(* Logix 5000 project; controller PLC_Safety vendor 1 type 14 code 148 rev 37.11; software revision 37.00 *)

TASK MainTask (continuous, watchdog 500 ms) : MainProgram
TASK SafetyTask (periodic, rate 20 ms, priority 10, watchdog 20 ms) : SafetyProgram

MODULES
   Local : vendor 1 type 14 code 148 (ICP 1, rev 37.11)
      Tarjeta_Ethernet : vendor 1 type 12 code 200 (ICP 0, Ethernet 10.12.143.10, rev 10.7, Input RPI 500 ms)
           Point_IO_Gabinete_6:2:I.1   // Push Button Gate 2 Reset
           Point_IO_Gabinete_6:2:I.2   // Push Button Gate 2 Open
         Kinetix_2 : vendor 1 type 37 code 48 (Ethernet 10.12.143.9, rev 7.1, MotionSync RPI 10 ms, MotionDiagnostics RPI 1 ms)
         Kinetix_1 : vendor 1 type 37 code 48 (Ethernet 10.12.143.8, rev 7.1, MotionDiagnostics RPI 1 ms, MotionSync RPI 10 ms)
         Cognex_3 : vendor 678 type 782 code 3585 (Ethernet 10.12.143.211, rev 1.1, StandardDataDriven RPI 20 ms)
         Fanuc_Brazo : vendor 8 type 140 code 34 (Ethernet 10.12.143.28, rev 2.4, StandardDataDriven RPI 20 ms)
              Fanuc_Brazo:I1.Input[2].4   // Input FANUC
              Fanuc_Brazo:I1.Input[3].0   // Input FANUC Rutina 5
              Fanuc_Brazo:I1.Input[3].1   // Input FANUC Rutina 6
              Fanuc_Brazo:I1.Input[3].2   // Input FANUC Rutina 7
              Fanuc_Brazo:O1.Output[0].3   // Cyle Stop - Abort
              Fanuc_Brazo:O1.Output[0]   // Fanuc Comands
              Fanuc_Brazo:O1.Output[2].0   // Strobe - Select
              Fanuc_Brazo:O1.Output[0].0   // Emergency Stop
              Fanuc_Brazo:O1.Output[0].1   // Hold
              Fanuc_Brazo:O1.Output[0].2   // Safe Speed
              Fanuc_Brazo:O1.Output[0].4   // Fault Reset
              Fanuc_Brazo:O1.Output[0].5   // Start
              Fanuc_Brazo:O1.Output[0].6   // Home
              Fanuc_Brazo:O1.Output[0].7   // Enable
              Fanuc_Brazo:O1.Output[1]   // Fanuc Routines
              Fanuc_Brazo:O1.Output[1].0   // No usar
              Fanuc_Brazo:O1.Output[1].1   // Routine 1 Base
              Fanuc_Brazo:O1.Output[1].2   // Routine 2 Centro
              Fanuc_Brazo:O1.Output[1].3   // Routine 3 Superior
              Fanuc_Brazo:O1.Output[1].4   // Routine 4 Assembly
              Fanuc_Brazo:O1.Output[2]   // Fanuc Strobe
         Fanuc_Delta : vendor 356 type 12 code 2 (Ethernet 10.12.143.47, rev 2.2, StandardDataDriven RPI 32 ms)
              Fanuc_Delta:I1.Input[0].1   // system ready
              Fanuc_Delta:I1.Input[0].0   // cmd enabled
              Fanuc_Delta:I1.Input[0].2   // prg running
              Fanuc_Delta:I1.Input[0].3   // prg paused
              Fanuc_Delta:I1.Input[0].4   // motion held
              Fanuc_Delta:I1.Input[0].5   // fault
              Fanuc_Delta:I1.Input[0].7   // tp enabled
              Fanuc_Delta:I1.Input[1].0   // batt alarm
              Fanuc_Delta:I1.Input[1].1   // busy
              Fanuc_Delta:I1.Input[1].2   // ack1
              Fanuc_Delta:I1.Input[1].3   // ack2
              Fanuc_Delta:I1.Input[1].4   // ack3
              Fanuc_Delta:I1.Input[1].5   // ack4
              Fanuc_Delta:I1.Input[1].6   // ack5
              Fanuc_Delta:I1.Input[1].7   // ack6
              Fanuc_Delta:I1.Input[2].0   // ack7
              Fanuc_Delta:I1.Input[2].1   // ack8
              Fanuc_Delta:I1.Input[2].2   // snack
              Fanuc_Delta:I1.Input[0].6   // at perch
              Fanuc_Delta:I1.Input[2].3   // reserved
              Fanuc_Delta:O1.Output[0].0   // IMSTP
              Fanuc_Delta:O1.Output[0].1   // hold
              Fanuc_Delta:O1.Output[0].2   // SFSPD
              Fanuc_Delta:O1.Output[0].3   // cycle stop
              Fanuc_Delta:O1.Output[0].4   // fault reset
              Fanuc_Delta:O1.Output[0].5   // start
              Fanuc_Delta:O1.Output[0].6   // Home
              Fanuc_Delta:O1.Output[0].7   // Enable
              Fanuc_Delta:O1.Output[1].0   // rsr1
              Fanuc_Delta:O1.Output[1].1   // rsr2
              Fanuc_Delta:O1.Output[1].2   // rsr3
              Fanuc_Delta:O1.Output[1].3   // rsr4
              Fanuc_Delta:O1.Output[1].4   // rsr5
              Fanuc_Delta:O1.Output[1].5   // rsr6
              Fanuc_Delta:O1.Output[1].6   // rsr7
              Fanuc_Delta:O1.Output[1].7   // rsr8
              Fanuc_Delta:O1.Output[2].0   // pns strobe
              Fanuc_Delta:O1.Output[2].1   // prod start
              Fanuc_Delta:O1.Output[2].5   // 22
              Fanuc_Delta:O1.Output[2].6   // 23
         Point_IO_Gabinete_3 : 1734-AENTR (Ethernet 10.12.143.42, rev 5.12, Output RPI 20 ms)
            Modulo_Input_Safety_3 : vendor 1 type 35 code 15 (PointIO 11, rev 2.2, Input RPI 10 ms)
                 Point_IO_Gabinete_3:11:I.Pt01Data   // Emergency Stop Conveyor 1 Normally Open
                 Point_IO_Gabinete_3:11:I.Pt00Data   // Emergency Stop Conveyor 1 Normally Close
                 Point_IO_Gabinete_3:11:I.Pt02Data   // SftyScanGab3 A (0=ObjDetec, 1=NoObjDetec)
                 Point_IO_Gabinete_3:11:I.Pt03Data   // SftyScanGab3 B (0=ObjDetec, 1=NoObjDetec)
            Modulo_Output_Safety_3 : vendor 1 type 35 code 16 (PointIO 12, rev 2.2, Input RPI 10 ms)
                 Point_IO_Gabinete_3:12:O.Pt01Data   // PowerFlex 1 Signal 2
                 Point_IO_Gabinete_3:12:O.Pt00Data   // PowerFlex 1 Signal 1
         Point_IO_Gabinete_1 : 1734-AENTR (Ethernet 10.12.143.40, rev 5.12, Output RPI 20 ms)
            Modulo_Output_Safety_1 : vendor 1 type 35 code 16 (PointIO 7, rev 2.2, Input RPI 10 ms)
                 Point_IO_Gabinete_1:7:O.Pt02Data   // GuardLock Gate 1
                 Point_IO_Gabinete_1:7:O.Pt01Data   // Kinetix 1 Signal 2
                 Point_IO_Gabinete_1:7:O.Pt00Data   // Kinetix 1 Signal 1
            Modulo_Input_Safety_1 : vendor 1 type 35 code 15 (PointIO 6, rev 2.2, Input RPI 10 ms)
                 Point_IO_Gabinete_1:6:I.Pt07Data   // Push Button Gate 1 Open
                 Point_IO_Gabinete_1:6:I.Pt05Data   // Guardlock Signal 2 Gate 1
                 Point_IO_Gabinete_1:6:I.Pt06Data   // Push Button Gate 1 Reset
                 Point_IO_Gabinete_1:6:I.Pt04Data   // GuardLock Signal 1 Gate 1
                 Point_IO_Gabinete_1:6:I.Pt01Data   // Emergency Stop 1 Normally Close
                 Point_IO_Gabinete_1:6:I.Pt00Data   // Emergency Stop 1 Normally Open
         Point_IO_Gabinete_2 : 1734-AENTR (Ethernet 10.12.143.41, rev 5.12, Output RPI 20 ms)   // Almacen Lado Derecho
            Modulo_Input_Safety_2 : vendor 1 type 35 code 15 (PointIO 6, rev 2.2, Input RPI 10 ms)
                 Point_IO_Gabinete_2:6:I.Pt06Data   // Push Button Process 2 Reset
                 Point_IO_Gabinete_2:6:I.Pt07Data   // Push Button Process 2 Start
                 Point_IO_Gabinete_2:6:I.Pt01Data   // Emergency Stop 2 Normally Close
                 Point_IO_Gabinete_2:6:I.Pt00Data   // Emergency Stop 2 Normally Open
            Modulo_Output_Safety_2 : vendor 1 type 35 code 16 (PointIO 7, rev 2.2, Input RPI 10 ms)
                 Point_IO_Gabinete_2:7:O.Pt01Data   // Kinetix 2 Signal 2
                 Point_IO_Gabinete_2:7:O.Pt00Data   // Kinetix 2 Signal 1
         Point_IO_Gabinete_4 : 1734-AENTR (Ethernet 10.12.143.43, rev 5.12, Output RPI 20 ms)   // Lado Izquierdo
            Modulo_Input_Safety_4 : vendor 1 type 35 code 15 (PointIO 11, rev 2.2, Input RPI 10 ms)
                 Point_IO_Gabinete_4:11:I.Pt02Data   // SftyScanGab4 A (0=ObjDetec, 1=NoObjDetec)
                 Point_IO_Gabinete_4:11:I.Pt03Data   // SftyScanGab4 B (0=ObjDetec, 1=NoObjDetec)
                 Point_IO_Gabinete_4:11:I.Pt01Data   // Emergency Stop Conveyor 2 Normally Open
                 Point_IO_Gabinete_4:11:I.Pt00Data   // Emergency Stop Conveyor 2 Normally Close
            Modulo_Output_Safety_4 : vendor 1 type 35 code 16 (PointIO 12, rev 2.2, Input RPI 10 ms)
                 Point_IO_Gabinete_4:12:O.Pt03Data   // Relay1 - ChB
                 Point_IO_Gabinete_4:12:O.Pt01Data   // Relay2 - ChB
                 Point_IO_Gabinete_4:12:O.Pt02Data   // Relay1 - ChA
                 Point_IO_Gabinete_4:12:O.Pt00Data   // Relay2 - ChA
                 Point_IO_Gabinete_4:12:O.Pt07Data   // PowerFlex 2 Signal 2
                 Point_IO_Gabinete_4:12:O.Pt06Data   // PowerFlex 2 Signal 1
         Point_IO_Gabinete_6 : 1734-AENTR (Ethernet 10.12.143.46, rev 5.11, Output RPI 20 ms)
            Modulo_Input_62 : 1734-IB8 (PointIO 2, rev 3.22)
            Modulo_Input_Safety_6 : vendor 1 type 35 code 15 (PointIO 4, rev 2.2, Input RPI 10 ms)
                 Point_IO_Gabinete_6:4:I.Pt01Data   // GuardLock Signal 2 Gate 2
                 Point_IO_Gabinete_6:4:I.Pt02Data   // Emergency Stop 3 Normally Close
                 Point_IO_Gabinete_6:4:I.Pt03Data   // Emergency Stop 3 Normally Open
                 Point_IO_Gabinete_6:4:I.Pt00Data   // GuardLock Signal 1 Gate 2
            Modulo_Output_Safety_6 : vendor 1 type 35 code 16 (PointIO 5, rev 2.2, Input RPI 10 ms)
                 Point_IO_Gabinete_6:5:O.Pt00Data   // GuardLock Gate 2
         PLC1 : vendor 1 type 14 code 235 (Ethernet 10.12.143.17, rev 37.11, $fc59bd35$ RPI 20 ms)
         PLC2 : vendor 1 type 14 code 235 (Ethernet 10.12.143.18, rev 37.11, $c2284200$ RPI 20 ms)
      @fcc730f7@:Partner : vendor 1 type 14 code 146 (ICP 2, rev 37.11)
END_MODULES

TYPE Auto_Data :
STRUCT
   Serial : STRING;
   Color : STRING;
   Peso : REAL;
   Llantas : DINT;
   Modo_Lujo : BOOL;
END_STRUCT
END_TYPE

VAR_GLOBAL   (* controller tags *)
   Axis_1 : AXIS_CIP_DRIVE;   // Storage 1
   Axis_2 : AXIS_CIP_DRIVE;   // Storage 2
   Data_From_PLC1 : DINT[20] := ([0] := 16781312);
   Data_From_PLC2 : DINT[20];
   Data_To_PLC1 : DINT[20] := ([0] := 1, [1] := 128); {produced}
        [0].13   // Tercera pieza recogida
        [0].12   // Segunda pieza recogida
        [0].11   // Primera pieza recogida
        [0].14   // Primera pieza para foto
        [0].15   // Segunda pieza para la foto
        [0].16   // Tercera pieza para la foto
   Data_To_PLC2 : DINT[20] := ([0] := 1, [2] := 1); {produced}
        [2].0   // E_stop_OK
   Display_Name : STRING;
   E_Stop_1_NC : ALIAS FOR Point_IO_Gabinete_1:6:I.Pt01Data;   // E Stop 1 Normally Close
   E_Stop_1_NO : ALIAS FOR Point_IO_Gabinete_1:6:I.Pt00Data;   // E Stop 1 Normally Open
   E_Stop_2_NC : ALIAS FOR Point_IO_Gabinete_2:6:I.Pt01Data;   // E Stop 2 Normally Close
   E_Stop_2_NO : ALIAS FOR Point_IO_Gabinete_2:6:I.Pt00Data;   // E Stop 2 Normally Open
   E_Stop_3_NC : ALIAS FOR Point_IO_Gabinete_6:4:I.Pt02Data;   // E Stop 3 Normally Close
   E_Stop_3_NO : ALIAS FOR Point_IO_Gabinete_6:4:I.Pt03Data;   // E Stop 3 Normally Open
   E_Stop_Conveyor_1_NC : ALIAS FOR Point_IO_Gabinete_3:11:I.Pt00Data;   // E Stop Conveyor 1 Normally Close
   E_Stop_Conveyor_1_NO : ALIAS FOR Point_IO_Gabinete_3:11:I.Pt01Data;   // E Stop Conveyor 1 Normally Open
   E_Stop_Conveyor_2_NC : ALIAS FOR Point_IO_Gabinete_4:11:I.Pt00Data;   // E Stop Conveyor 2 Normally Close
   E_Stop_Conveyor_2_NO : ALIAS FOR Point_IO_Gabinete_4:11:I.Pt01Data;   // E Stop Conveyor 2 Normally Open
   E_Stop_OK : BOOL := 1;
   Fanuc_E_Stop_SFTY : BOOL := 1;
   Fanuc_E_Stop_STD : BOOL := 1;
   Fanuc_Fault_Reset_SFTY : BOOL;
   Fanuc_Fault_Reset_STD : BOOL;
   Gate_1_Open_SFTY : ALIAS FOR Point_IO_Gabinete_1:6:I.Pt07Data;   // Push Button Gate 1 Open
   Gate_1_Reset_SFTY : ALIAS FOR Point_IO_Gabinete_1:6:I.Pt06Data;   // Push Button Gate 1 Reset
   Gate_2_Open_SFTY : BOOL;   // Push Button Gate 2 Open
   Gate_2_Open_STD : BOOL;   // Push Button Gate 2 Open
   Gate_2_Reset_SFTY : BOOL;   // Push Button Gate 2 Reset
   Gate_2_Reset_STD : BOOL;   // Push Button Gate 2 Reset
   Manual_SFTY : BOOL := 1;
   Manual_STD : BOOL := 1;
   Motion : MOTION_GROUP;
   Process_1_Reset_SFTY : BOOL;   // Push Button Process 1 Reset
   Process_1_Reset_STD : BOOL;   // Push Button Process 1 Reset
   Process_2_Reset_SFTY : ALIAS FOR Point_IO_Gabinete_2:6:I.Pt06Data;   // Push Button Process 2 Reset
   Process_2_Start_SFTY : ALIAS FOR Point_IO_Gabinete_2:6:I.Pt07Data;   // Push Button Porcess 2 Start
   Reset_General : BOOL;
   S1_Height_1 : BOOL;
   S1_Height_2 : BOOL;
   S1_Height_3 : BOOL;
   S1_Height_4 : BOOL;
   S1_Height_5 : BOOL;
   S1_Height_6 : BOOL;
   S1_Height_Conveyor_1 : BOOL;
   S1_Height_Conveyor_2 : BOOL;
   S1_Storage_On : BOOL;
   Safety_OK : BOOL := 1;
   Start_Button_1_Squence : BOOL;
END_VAR

PROGRAM MainProgram   (* main routine R00_Main_Routine *)
VAR
   Assembly_Step : DINT;
   Contador_num_pza : COUNTER;
   Contador_pza_aprove : COUNTER := (CU := 1, DN := 1);
   Contador_pza_rechazada : COUNTER := (DN := 1);
   Counter_Parts : COUNTER := (ACC := 2, CU := 1, DN := 1);   // Trazabilidad
   Done_cicle : BOOL;
   Error_Cam : DINT;
   FANUC_R1 : BOOL := 1;
   FANUC_R2 : BOOL;
   FANUC_R3 : BOOL;
   FANUC_R4 : BOOL;
   Fanuc_Strobe : BOOL;
   HMI_Cognex_1 : DINT;   // HMI
   HMI_Cognex_2 : DINT;   // HMI
   HMI_Cognex_medio : DINT;   // HMI
   HMI_Fanucbrazo : DINT := 516;   // HMI
   HMI_Fanucdelta : DINT := 516;   // HMI
   HMI_Fcognex1 : BOOL;   // HMI
   HMI_Fcognex2 : BOOL;   // HMI
   HMI_Fcognexmedio : BOOL;   // HMI
   HMI_Ffanucbrazo : BOOL := 1;   // HMI
   HMI_Ffanucdelta : BOOL := 1;   // HMI
   HMI_Fplc1 : BOOL;   // HMI
   HMI_Fplc2 : BOOL;   // HMI
   HMI_Fplcseguridad : BOOL;   // HMI
   HMI_kinetix1 : BOOL;   // HMI
   HMI_kinetix2 : BOOL;
   HMI_Kinetix_1 : DINT;   // HMI
   HMI_Kinetix_2 : DINT;
   HMI_PLC1 : DINT;   // HMI
   HMI_PLC2 : DINT;   // HMI
   HMI_PLC_Seguridad : DINT;   // HMI
   HMI_PointIO1 : BOOL;   // HMI
   HMI_PointIO2 : BOOL;
   HMI_PointIO3 : BOOL;
   HMI_PointIO4 : BOOL;
   HMI_PointIO6 : BOOL;
   HMI_PointIO_1 : DINT;   // HMI
   HMI_PointIO_2 : DINT;
   HMI_PointIO_3 : DINT;
   HMI_PointIO_4 : DINT;
   HMI_PointIO_6 : DINT;
   HMI_R_Axis_Y_Negative : BOOL;
   HMI_R_Axis_Y_Positive : BOOL;
   HMI_R_cognex1 : BOOL := 1;
   HMI_R_cognex2 : BOOL;
   HMI_R_con2OFF : BOOL;
   HMI_R_con2ON : BOOL;
   HMI_R_Conveyor_OFF : BOOL;
   HMI_R_Conveyor_ON : BOOL;
   HMI_R_Gripper_Close : BOOL;
   HMI_R_Gripper_Open : BOOL;
   HMI_R_Height_4_1 : BOOL;
   HMI_R_Height_4_2 : BOOL;
   HMI_R_Height_5_1 : BOOL;
   HMI_R_Height_5_2 : BOOL;
   HMI_R_Height_6_1 : BOOL;
   HMI_R_Height_6_2 : BOOL;
   HMI_R_lane1 : BOOL;
   HMI_R_lane1_c2 : BOOL;
   HMI_R_lane2 : BOOL;
   HMI_R_lane2_c2 : BOOL;
   HMI_R_onoff : BOOL := 1;
   HMI_R_PF1 : BOOL;
   HMI_R_PF2 : BOOL;
   HMI_R_pis0 : BOOL;
   HMI_R_pis1 : BOOL;
   HMI_R_pis2 : BOOL;
   HMI_R_pis3 : BOOL;
   HMI_R_pis4 : BOOL;
   HMI_R_pis5 : BOOL;
   HMI_R_pis6 : BOOL;
   HMI_R_pis7 : BOOL;
   HMI_R_pis8 : BOOL;
   HMI_R_pis9 : BOOL;
   HMI_R_Turn_Conveyor : BOOL;
   HMI_R_Turn_Storage : BOOL;
   HMI_S_Axis_Y_Negative : BOOL;
   HMI_S_Axis_Y_Positive : BOOL;
   HMI_S_cognex1 : BOOL := 1;
   HMI_S_cognex2 : BOOL;
   HMI_S_con2Off : BOOL;
   HMI_S_con2ON : BOOL;
   HMI_S_Conveyor_OFF : BOOL;
   HMI_S_Conveyor_ON : BOOL;
   HMI_S_Gripper_Close : BOOL;
   HMI_S_Gripper_Open : BOOL;
   HMI_S_Height_4_1 : BOOL;
   HMI_S_Height_4_2 : BOOL;
   HMI_S_Height_5_1 : BOOL;
   HMI_S_Height_5_2 : BOOL;
   HMI_S_Height_6_1 : BOOL;
   HMI_S_Height_6_2 : BOOL;
   HMI_S_lane1 : BOOL;
   HMI_S_lane1_c2 : BOOL;
   HMI_S_lane2 : BOOL;
   HMI_S_lane2_c2 : BOOL;
   HMI_S_onoff : BOOL := 1;
   HMI_S_PF1 : BOOL;
   HMI_S_PF2 : BOOL;
   HMI_S_pis0 : BOOL;
   HMI_S_pis1 : BOOL;
   HMI_S_pis2 : BOOL;
   HMI_S_pis3 : BOOL;
   HMI_S_pis4 : BOOL;
   HMI_S_pis5 : BOOL;
   HMI_S_pis6 : BOOL;
   HMI_S_pis7 : BOOL;
   HMI_S_pis8 : BOOL;
   HMI_S_pis9 : BOOL;
   HMI_S_Turn_Conveyor : BOOL;
   HMI_S_Turn_Storage : BOOL;
   HMI_Switch1 : BOOL;
   HMI_Switch2 : BOOL;
   HMI_Switch3 : BOOL := 1;
   HMI_Switch4 : BOOL;
   HMI_Switch5 : BOOL := 1;
   OSF_Fault_Reset_Fanuc : BOOL;
   Part : REAL := 1.0;
   Piece_Approved : BOOL := 1;
   Piece_Base : BOOL := 1;
   Piece_Coil : BOOL;
   Piece_Rejected : BOOL;
   Piece_Upper : BOOL;
   Process_Result : BOOL;
   Result_OneShot : BOOL;
   S1_Height_4_Number_2 : BOOL;
   S1_Height_5_Number_2 : BOOL;
   S1_Height_6_Number_2 : BOOL;
   S1_MAM_Height_1 : MOTION_INSTRUCTION := (FLAGS := 33554432);
   S1_MAM_Height_2 : MOTION_INSTRUCTION := (FLAGS := 33554432);
   S1_MAM_Height_3 : MOTION_INSTRUCTION := (FLAGS := 33554432);
   S1_MAM_Height_4 : MOTION_INSTRUCTION := (FLAGS := 33554432);
   S1_MAM_Height_4_Number_2 : MOTION_INSTRUCTION := (FLAGS := 33554432);
   S1_MAM_Height_5 : MOTION_INSTRUCTION := (FLAGS := 33554432);
   S1_MAM_Height_5_Number_2 : MOTION_INSTRUCTION := (FLAGS := 33554432);
   S1_MAM_Height_6 : MOTION_INSTRUCTION := (FLAGS := 33554432);
   S1_MAM_Height_6_Number_2 : MOTION_INSTRUCTION := (FLAGS := 33554432);
   S1_MAM_Height_Conveyor_1 : MOTION_INSTRUCTION := (FLAGS := 33554432);
   S1_MAM_Height_Conveyor_2 : MOTION_INSTRUCTION := (FLAGS := 33554432);
   S1_MSO_Storage : MOTION_INSTRUCTION := (FLAGS := 33554432);
   S1_Sensor_Height_1 : BOOL;
   S1_Sensor_Height_2 : BOOL;
   S1_Sensor_Height_3 : BOOL;
   S1_Sensor_Height_4 : BOOL;
   S1_Sensor_Height_4_Number_2 : BOOL;
   S1_Sensor_Height_5 : BOOL;
   S1_Sensor_Height_5_Number_2 : BOOL;
   S1_Sensor_Height_6 : BOOL;
   S1_Sensor_Height_6_Number_2 : BOOL;
   S1_Sensor_Height_Conveyor_1 : BOOL;
   S1_Sensor_Height_Conveyor_2 : BOOL;
   S2_Height_1 : BOOL;
   S2_Height_2 : BOOL;
   S2_Height_3 : BOOL;
   S2_Height_4 : BOOL;
   S2_Height_4_Number_2 : BOOL;
   S2_Height_5 : BOOL;
   S2_Height_5_Number_2 : BOOL;
   S2_Height_6 : BOOL;
   S2_Height_Conveyor_1 : BOOL;
   S2_Height_Conveyor_2 : BOOL;
   S2_MAM_Height_1 : MOTION_INSTRUCTION;
   S2_MAM_Height_2 : MOTION_INSTRUCTION;
   S2_MAM_Height_3 : MOTION_INSTRUCTION;
   S2_MAM_Height_4 : MOTION_INSTRUCTION;
   S2_MAM_Height_4_Number_2 : MOTION_INSTRUCTION;
   S2_MAM_Height_5 : MOTION_INSTRUCTION;
   S2_MAM_Height_5_Number_2 : MOTION_INSTRUCTION;
   S2_MAM_Height_6 : MOTION_INSTRUCTION;
   S2_MAM_Height_Conveyor_1 : MOTION_INSTRUCTION;
   S2_MAM_Height_Conveyor_2 : MOTION_INSTRUCTION;
   S2_MSO_Storage : MOTION_INSTRUCTION;
   S2_Sensor_Height_1 : BOOL;
   S2_Sensor_Height_2 : BOOL;
   S2_Sensor_Height_3 : BOOL;
   S2_Sensor_Height_4 : BOOL;
   S2_Sensor_Height_5 : BOOL;
   S2_Sensor_Height_6 : BOOL;
   S2_Sensor_Height_Conveyor_1 : BOOL;
   S2_Sensor_Height_Conveyor_2 : BOOL;
   S2_Storage_On : BOOL;
   Sensor_FANUC_R1 : BOOL;
   Sensor_FANUC_R2 : BOOL;
   Sensor_FANUC_R3 : BOOL;
   Sensor_FANUC_R4 : BOOL;
   Start_Button_1_Secuencia : BOOL;
   Start_Button_2_Secuencia : BOOL;
   Start_Button_3_Secuencia : BOOL;
   Stop_general : BOOL;
   Trigger_Cognex_3 : BOOL;
END_VAR

ROUTINE HMI_Manual_Safety   (* ladder *)
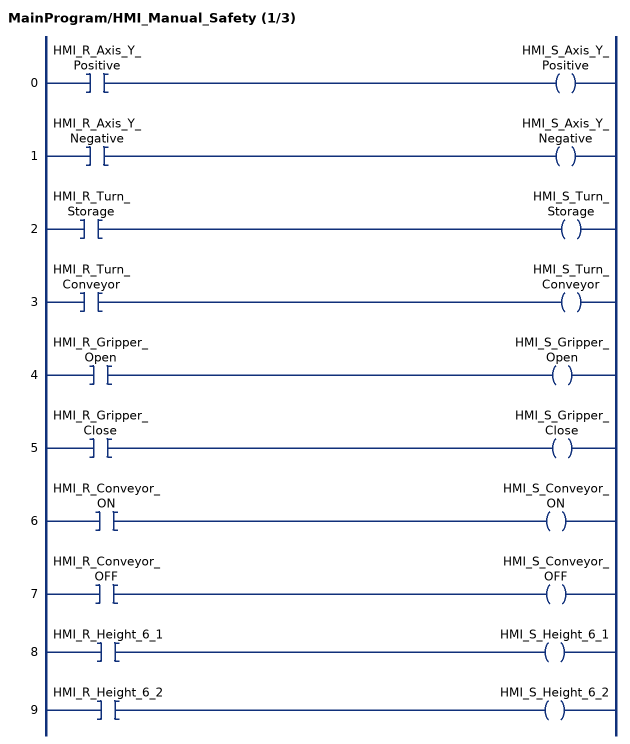
   0: XIC(HMI_R_Axis_Y_Positive)OTE(HMI_S_Axis_Y_Positive);
   1: XIC(HMI_R_Axis_Y_Negative)OTE(HMI_S_Axis_Y_Negative);
   2: XIC(HMI_R_Turn_Storage)OTE(HMI_S_Turn_Storage);
   3: XIC(HMI_R_Turn_Conveyor)OTE(HMI_S_Turn_Conveyor);
   4: XIC(HMI_R_Gripper_Open)OTE(HMI_S_Gripper_Open);
   5: XIC(HMI_R_Gripper_Close)OTE(HMI_S_Gripper_Close);
   6: XIC(HMI_R_Conveyor_ON)OTE(HMI_S_Conveyor_ON);
   7: XIC(HMI_R_Conveyor_OFF)OTE(HMI_S_Conveyor_OFF);
   8: XIC(HMI_R_Height_6_1)OTE(HMI_S_Height_6_1);
   9: XIC(HMI_R_Height_6_2)OTE(HMI_S_Height_6_2);
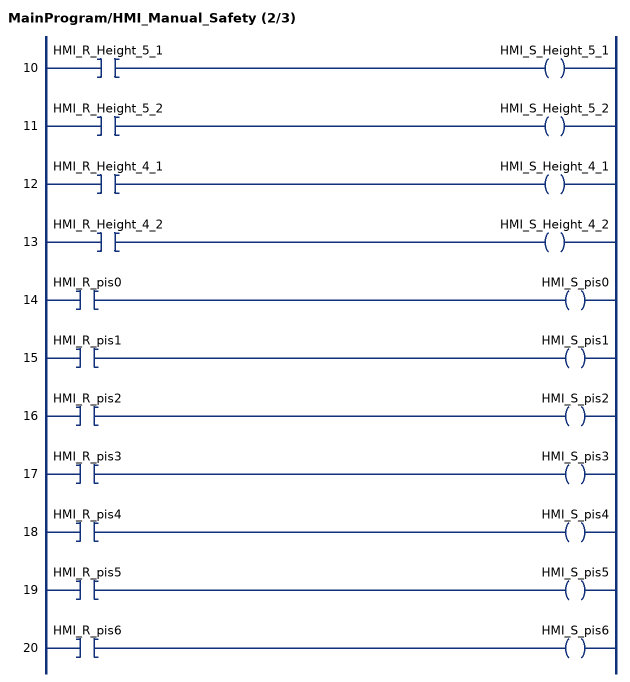
   10: XIC(HMI_R_Height_5_1)OTE(HMI_S_Height_5_1);
   11: XIC(HMI_R_Height_5_2)OTE(HMI_S_Height_5_2);
   12: XIC(HMI_R_Height_4_1)OTE(HMI_S_Height_4_1);
   13: XIC(HMI_R_Height_4_2)OTE(HMI_S_Height_4_2);
   14: XIC(HMI_R_pis0)OTE(HMI_S_pis0);
   15: XIC(HMI_R_pis1)OTE(HMI_S_pis1);
   16: XIC(HMI_R_pis2)OTE(HMI_S_pis2);
   17: XIC(HMI_R_pis3)OTE(HMI_S_pis3);
   18: XIC(HMI_R_pis4)OTE(HMI_S_pis4);
   19: XIC(HMI_R_pis5)OTE(HMI_S_pis5);
   20: XIC(HMI_R_pis6)OTE(HMI_S_pis6);
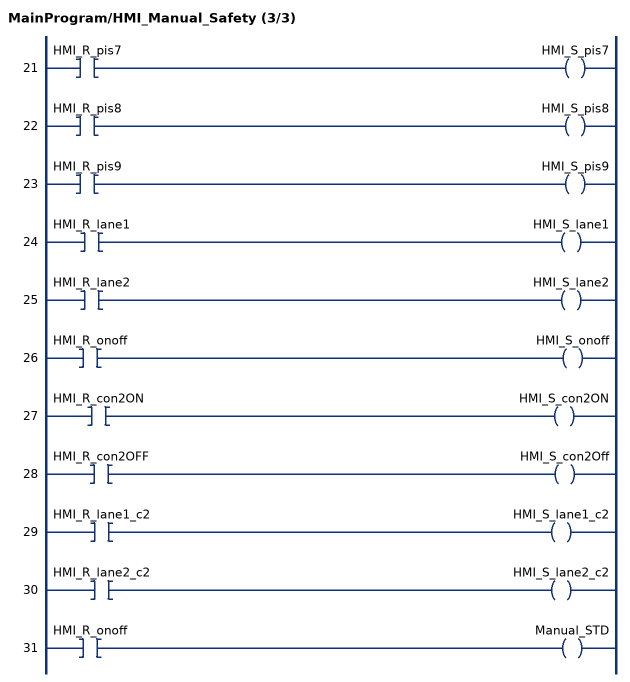
   21: XIC(HMI_R_pis7)OTE(HMI_S_pis7);
   22: XIC(HMI_R_pis8)OTE(HMI_S_pis8);
   23: XIC(HMI_R_pis9)OTE(HMI_S_pis9);
   24: XIC(HMI_R_lane1)OTE(HMI_S_lane1);
   25: XIC(HMI_R_lane2)OTE(HMI_S_lane2);
   26: XIC(HMI_R_onoff)OTE(HMI_S_onoff);
   27: XIC(HMI_R_con2ON)OTE(HMI_S_con2ON);
   28: XIC(HMI_R_con2OFF)OTE(HMI_S_con2Off);
   29: XIC(HMI_R_lane1_c2)OTE(HMI_S_lane1_c2);
   30: XIC(HMI_R_lane2_c2)OTE(HMI_S_lane2_c2);
   31: XIC(HMI_R_onoff)OTE(Manual_STD);
END_ROUTINE

ROUTINE R00_Main_Routine   (* ladder *)
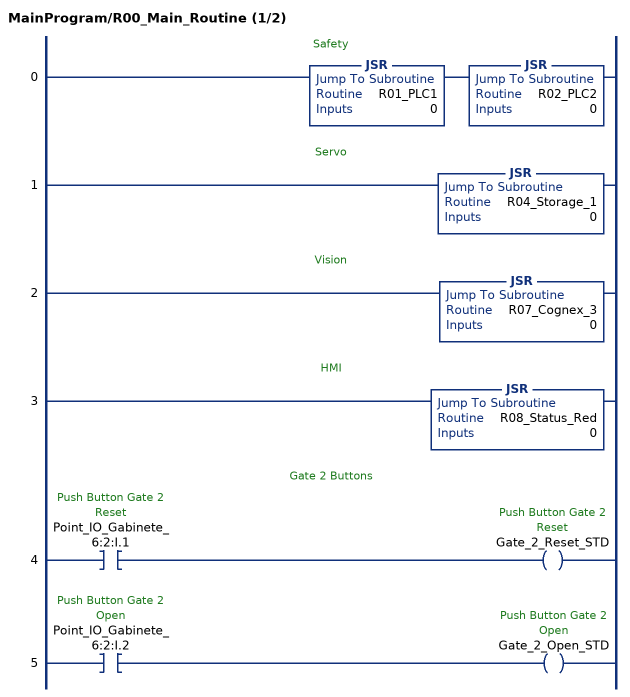
   // Safety
   0: JSR(R01_PLC1,0)JSR(R02_PLC2,0);
   // Servo
   1: JSR(R04_Storage_1,0);
   // Vision
   2: JSR(R07_Cognex_3,0);
   // HMI
   3: JSR(R08_Status_Red,0);
   // Gate 2 Buttons
   4: XIC(Point_IO_Gabinete_6:2:I.1)OTE(Gate_2_Reset_STD);
   5: XIC(Point_IO_Gabinete_6:2:I.2)OTE(Gate_2_Open_STD);
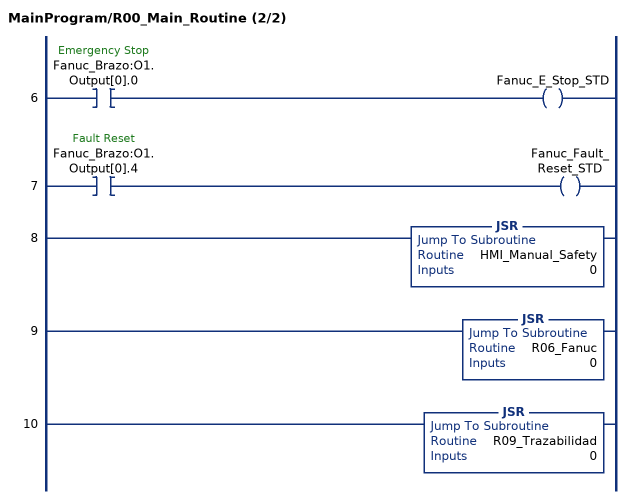
   6: XIC(Fanuc_Brazo:O1.Output[0].0)OTE(Fanuc_E_Stop_STD);
   7: XIC(Fanuc_Brazo:O1.Output[0].4)OTE(Fanuc_Fault_Reset_STD);
   8: JSR(HMI_Manual_Safety,0);
   9: JSR(R06_Fanuc,0);
   10: JSR(R09_Trazabilidad,0);
END_ROUTINE

ROUTINE R01_PLC1   (* ladder *)
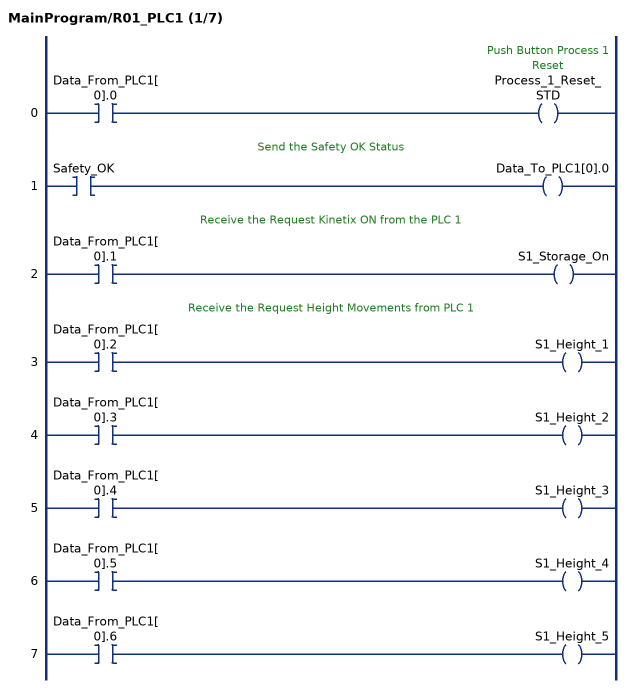
   0: XIC(Data_From_PLC1[0].0)OTE(Process_1_Reset_STD);
   // Send the Safety OK Status
   1: XIC(Safety_OK)OTE(Data_To_PLC1[0].0);
   // Receive the Request Kinetix ON from the PLC 1
   2: XIC(Data_From_PLC1[0].1)OTE(S1_Storage_On);
   // Receive the Request Height Movements from PLC 1
   3: XIC(Data_From_PLC1[0].2)OTE(S1_Height_1);
   4: XIC(Data_From_PLC1[0].3)OTE(S1_Height_2);
   5: XIC(Data_From_PLC1[0].4)OTE(S1_Height_3);
   6: XIC(Data_From_PLC1[0].5)OTE(S1_Height_4);
   7: XIC(Data_From_PLC1[0].6)OTE(S1_Height_5);
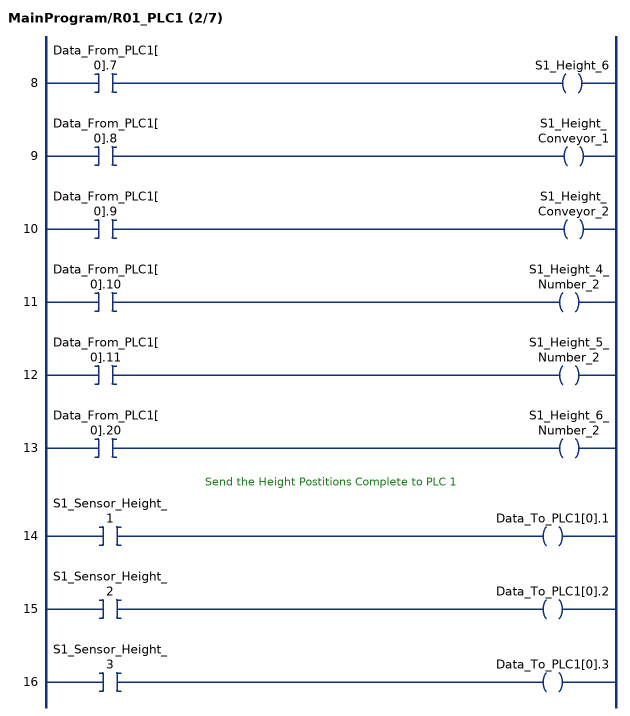
   8: XIC(Data_From_PLC1[0].7)OTE(S1_Height_6);
   9: XIC(Data_From_PLC1[0].8)OTE(S1_Height_Conveyor_1);
   10: XIC(Data_From_PLC1[0].9)OTE(S1_Height_Conveyor_2);
   11: XIC(Data_From_PLC1[0].10)OTE(S1_Height_4_Number_2);
   12: XIC(Data_From_PLC1[0].11)OTE(S1_Height_5_Number_2);
   13: XIC(Data_From_PLC1[0].20)OTE(S1_Height_6_Number_2);
   // Send the Height Postitions Complete to PLC 1
   14: XIC(S1_Sensor_Height_1)OTE(Data_To_PLC1[0].1);
   15: XIC(S1_Sensor_Height_2)OTE(Data_To_PLC1[0].2);
   16: XIC(S1_Sensor_Height_3)OTE(Data_To_PLC1[0].3);
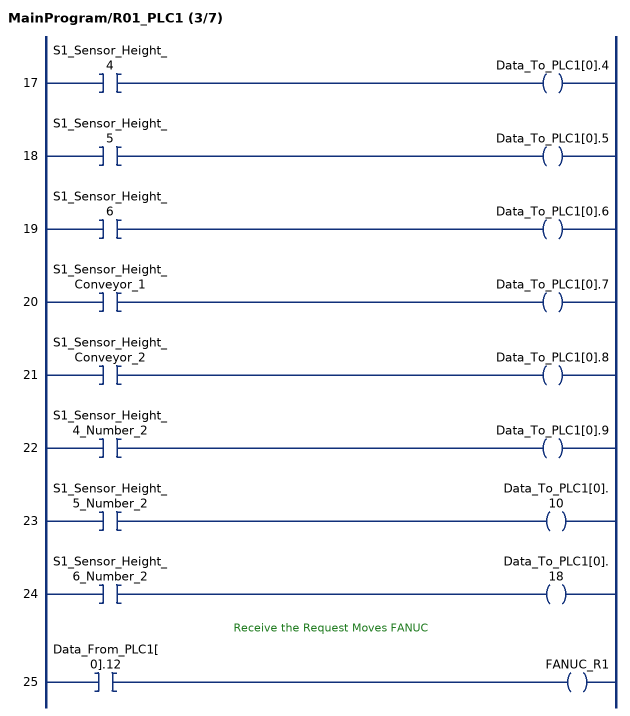
   17: XIC(S1_Sensor_Height_4)OTE(Data_To_PLC1[0].4);
   18: XIC(S1_Sensor_Height_5)OTE(Data_To_PLC1[0].5);
   19: XIC(S1_Sensor_Height_6)OTE(Data_To_PLC1[0].6);
   20: XIC(S1_Sensor_Height_Conveyor_1)OTE(Data_To_PLC1[0].7);
   21: XIC(S1_Sensor_Height_Conveyor_2)OTE(Data_To_PLC1[0].8);
   22: XIC(S1_Sensor_Height_4_Number_2)OTE(Data_To_PLC1[0].9);
   23: XIC(S1_Sensor_Height_5_Number_2)OTE(Data_To_PLC1[0].10);
   24: XIC(S1_Sensor_Height_6_Number_2)OTE(Data_To_PLC1[0].18);
   // Receive the Request Moves FANUC
   25: XIC(Data_From_PLC1[0].12)OTE(FANUC_R1);
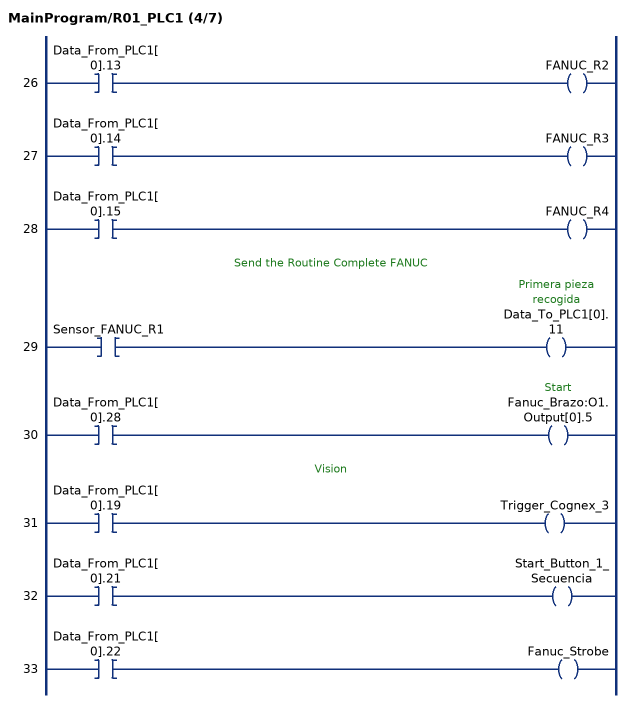
   26: XIC(Data_From_PLC1[0].13)OTE(FANUC_R2);
   27: XIC(Data_From_PLC1[0].14)OTE(FANUC_R3);
   28: XIC(Data_From_PLC1[0].15)OTE(FANUC_R4);
   // Send the Routine Complete FANUC
   29: XIC(Sensor_FANUC_R1)OTE(Data_To_PLC1[0].11);
   30: XIC(Data_From_PLC1[0].28)OTE(Fanuc_Brazo:O1.Output[0].5);
   // Vision
   31: XIC(Data_From_PLC1[0].19)OTE(Trigger_Cognex_3);
   32: XIC(Data_From_PLC1[0].21)OTE(Start_Button_1_Secuencia);
   33: XIC(Data_From_PLC1[0].22)OTE(Fanuc_Strobe);
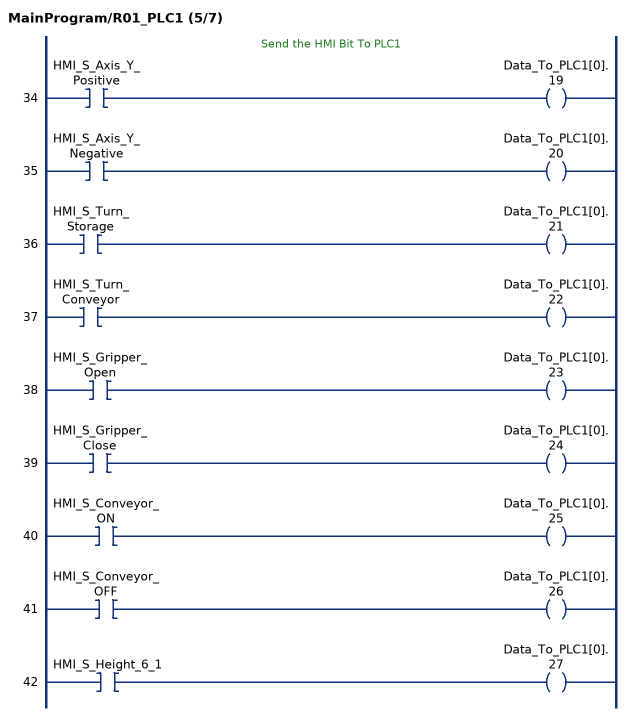
   // Send the HMI Bit To PLC1
   34: XIC(HMI_S_Axis_Y_Positive)OTE(Data_To_PLC1[0].19);
   35: XIC(HMI_S_Axis_Y_Negative)OTE(Data_To_PLC1[0].20);
   36: XIC(HMI_S_Turn_Storage)OTE(Data_To_PLC1[0].21);
   37: XIC(HMI_S_Turn_Conveyor)OTE(Data_To_PLC1[0].22);
   38: XIC(HMI_S_Gripper_Open)OTE(Data_To_PLC1[0].23);
   39: XIC(HMI_S_Gripper_Close)OTE(Data_To_PLC1[0].24);
   40: XIC(HMI_S_Conveyor_ON)OTE(Data_To_PLC1[0].25);
   41: XIC(HMI_S_Conveyor_OFF)OTE(Data_To_PLC1[0].26);
   42: XIC(HMI_S_Height_6_1)OTE(Data_To_PLC1[0].27);
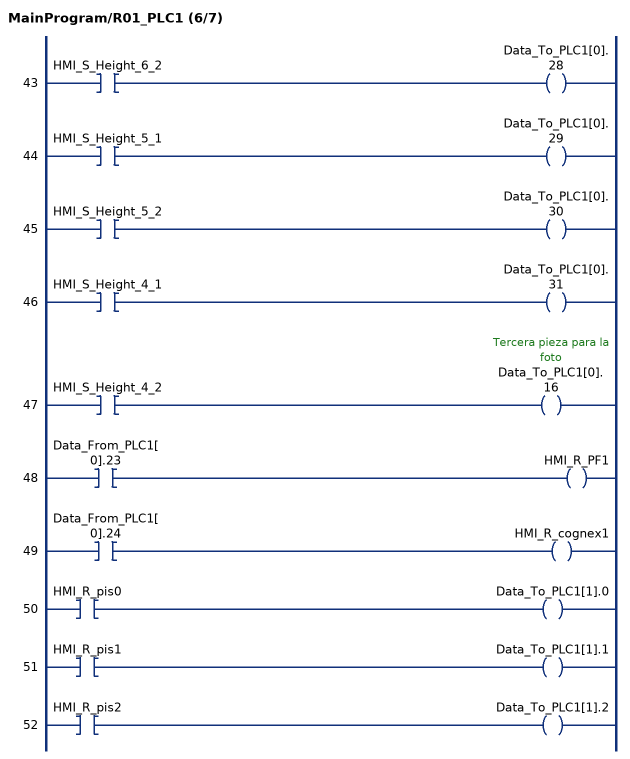
   43: XIC(HMI_S_Height_6_2)OTE(Data_To_PLC1[0].28);
   44: XIC(HMI_S_Height_5_1)OTE(Data_To_PLC1[0].29);
   45: XIC(HMI_S_Height_5_2)OTE(Data_To_PLC1[0].30);
   46: XIC(HMI_S_Height_4_1)OTE(Data_To_PLC1[0].31);
   47: XIC(HMI_S_Height_4_2)OTE(Data_To_PLC1[0].16);
   48: XIC(Data_From_PLC1[0].23)OTE(HMI_R_PF1);
   49: XIC(Data_From_PLC1[0].24)OTE(HMI_R_cognex1);
   50: XIC(HMI_R_pis0)OTE(Data_To_PLC1[1].0);
   51: XIC(HMI_R_pis1)OTE(Data_To_PLC1[1].1);
   52: XIC(HMI_R_pis2)OTE(Data_To_PLC1[1].2);
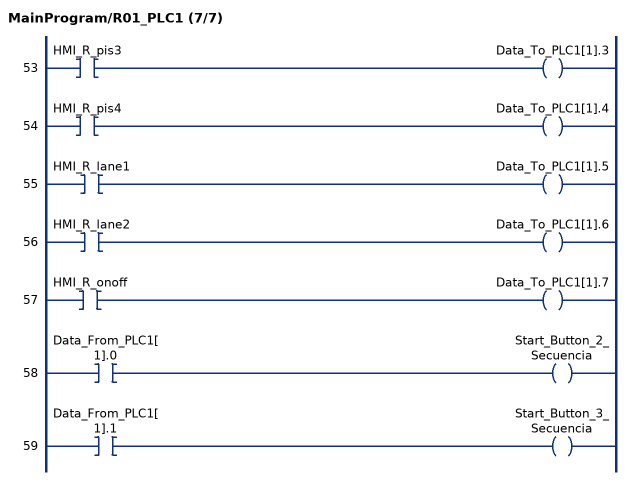
   53: XIC(HMI_R_pis3)OTE(Data_To_PLC1[1].3);
   54: XIC(HMI_R_pis4)OTE(Data_To_PLC1[1].4);
   55: XIC(HMI_R_lane1)OTE(Data_To_PLC1[1].5);
   56: XIC(HMI_R_lane2)OTE(Data_To_PLC1[1].6);
   57: XIC(HMI_R_onoff)OTE(Data_To_PLC1[1].7);
   58: XIC(Data_From_PLC1[1].0)OTE(Start_Button_2_Secuencia);
   59: XIC(Data_From_PLC1[1].1)OTE(Start_Button_3_Secuencia);
END_ROUTINE

ROUTINE R02_PLC2   (* ladder *)
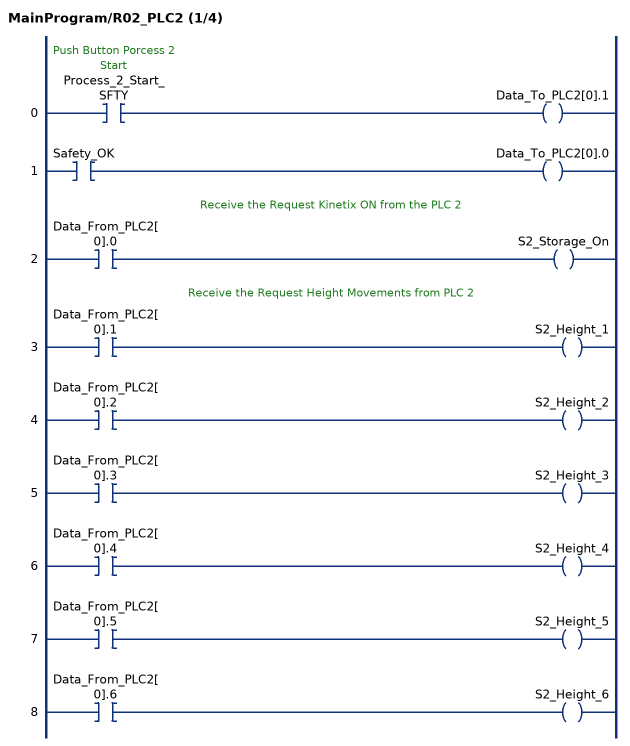
   0: XIC(Process_2_Start_SFTY)OTE(Data_To_PLC2[0].1);
   1: XIC(Safety_OK)OTE(Data_To_PLC2[0].0);
   // Receive the Request Kinetix ON from the PLC 2
   2: XIC(Data_From_PLC2[0].0)OTE(S2_Storage_On);
   // Receive the Request Height Movements from PLC 2
   3: XIC(Data_From_PLC2[0].1)OTE(S2_Height_1);
   4: XIC(Data_From_PLC2[0].2)OTE(S2_Height_2);
   5: XIC(Data_From_PLC2[0].3)OTE(S2_Height_3);
   6: XIC(Data_From_PLC2[0].4)OTE(S2_Height_4);
   7: XIC(Data_From_PLC2[0].5)OTE(S2_Height_5);
   8: XIC(Data_From_PLC2[0].6)OTE(S2_Height_6);
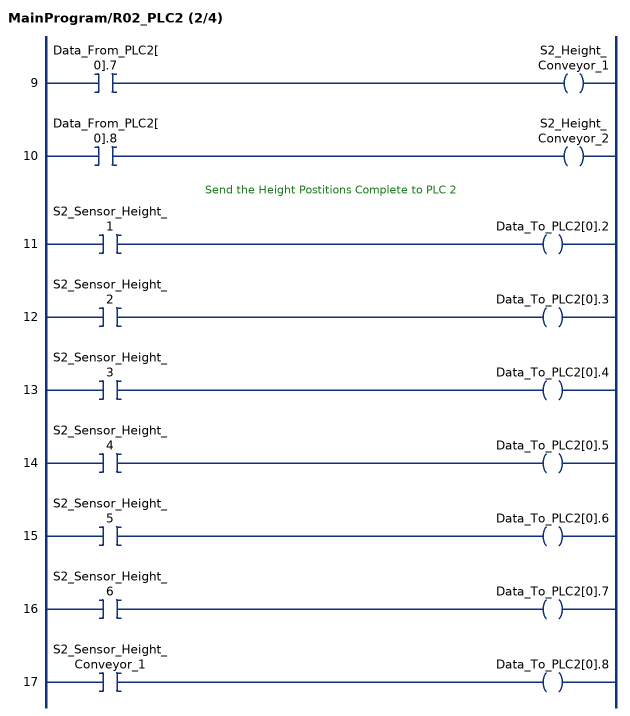
   9: XIC(Data_From_PLC2[0].7)OTE(S2_Height_Conveyor_1);
   10: XIC(Data_From_PLC2[0].8)OTE(S2_Height_Conveyor_2);
   // Send the Height Postitions Complete to PLC 2
   11: XIC(S2_Sensor_Height_1)OTE(Data_To_PLC2[0].2);
   12: XIC(S2_Sensor_Height_2)OTE(Data_To_PLC2[0].3);
   13: XIC(S2_Sensor_Height_3)OTE(Data_To_PLC2[0].4);
   14: XIC(S2_Sensor_Height_4)OTE(Data_To_PLC2[0].5);
   15: XIC(S2_Sensor_Height_5)OTE(Data_To_PLC2[0].6);
   16: XIC(S2_Sensor_Height_6)OTE(Data_To_PLC2[0].7);
   17: XIC(S2_Sensor_Height_Conveyor_1)OTE(Data_To_PLC2[0].8);
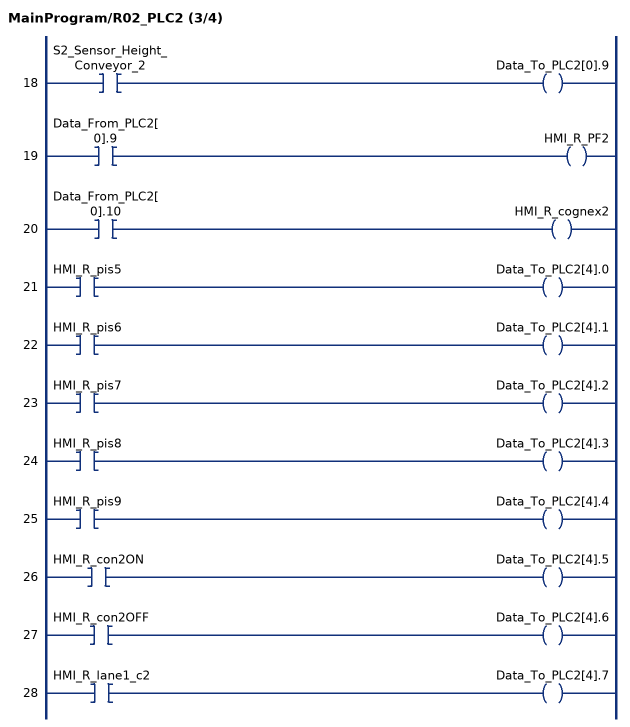
   18: XIC(S2_Sensor_Height_Conveyor_2)OTE(Data_To_PLC2[0].9);
   19: XIC(Data_From_PLC2[0].9)OTE(HMI_R_PF2);
   20: XIC(Data_From_PLC2[0].10)OTE(HMI_R_cognex2);
   21: XIC(HMI_R_pis5)OTE(Data_To_PLC2[4].0);
   22: XIC(HMI_R_pis6)OTE(Data_To_PLC2[4].1);
   23: XIC(HMI_R_pis7)OTE(Data_To_PLC2[4].2);
   24: XIC(HMI_R_pis8)OTE(Data_To_PLC2[4].3);
   25: XIC(HMI_R_pis9)OTE(Data_To_PLC2[4].4);
   26: XIC(HMI_R_con2ON)OTE(Data_To_PLC2[4].5);
   27: XIC(HMI_R_con2OFF)OTE(Data_To_PLC2[4].6);
   28: XIC(HMI_R_lane1_c2)OTE(Data_To_PLC2[4].7);
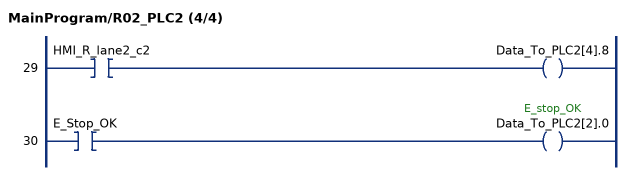
   29: XIC(HMI_R_lane2_c2)OTE(Data_To_PLC2[4].8);
   30: XIC(E_Stop_OK)OTE(Data_To_PLC2[2].0);
END_ROUTINE

ROUTINE R04_Storage_1   (* ladder *)
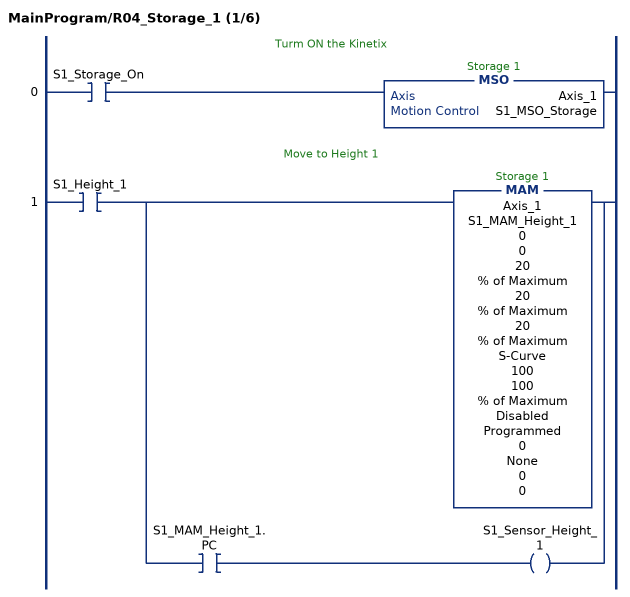
   // Turm ON the Kinetix
   0: XIC(S1_Storage_On)MSO(Axis_1,S1_MSO_Storage);
   // Move to Height 1
   1: XIC(S1_Height_1)[MAM(Axis_1,S1_MAM_Height_1,0,0,20,% of Maximum,20,% of Maximum,20,% of Maximum,S-Curve,100,100,% of Maximum,Disabled,Programmed,0,None,0,0) ,XIC(S1_MAM_Height_1.PC) OTE(S1_Sensor_Height_1) ];
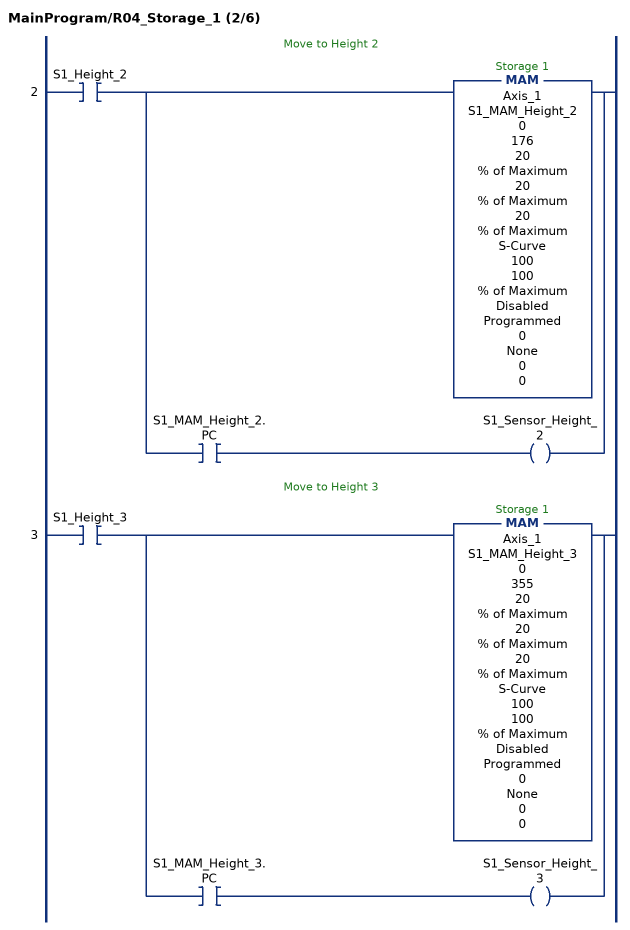
   // Move to Height 2
   2: XIC(S1_Height_2)[MAM(Axis_1,S1_MAM_Height_2,0,176,20,% of Maximum,20,% of Maximum,20,% of Maximum,S-Curve,100,100,% of Maximum,Disabled,Programmed,0,None,0,0) ,XIC(S1_MAM_Height_2.PC) OTE(S1_Sensor_Height_2) ];
   // Move to Height 3
   3: XIC(S1_Height_3)[MAM(Axis_1,S1_MAM_Height_3,0,355,20,% of Maximum,20,% of Maximum,20,% of Maximum,S-Curve,100,100,% of Maximum,Disabled,Programmed,0,None,0,0) ,XIC(S1_MAM_Height_3.PC) OTE(S1_Sensor_Height_3) ];
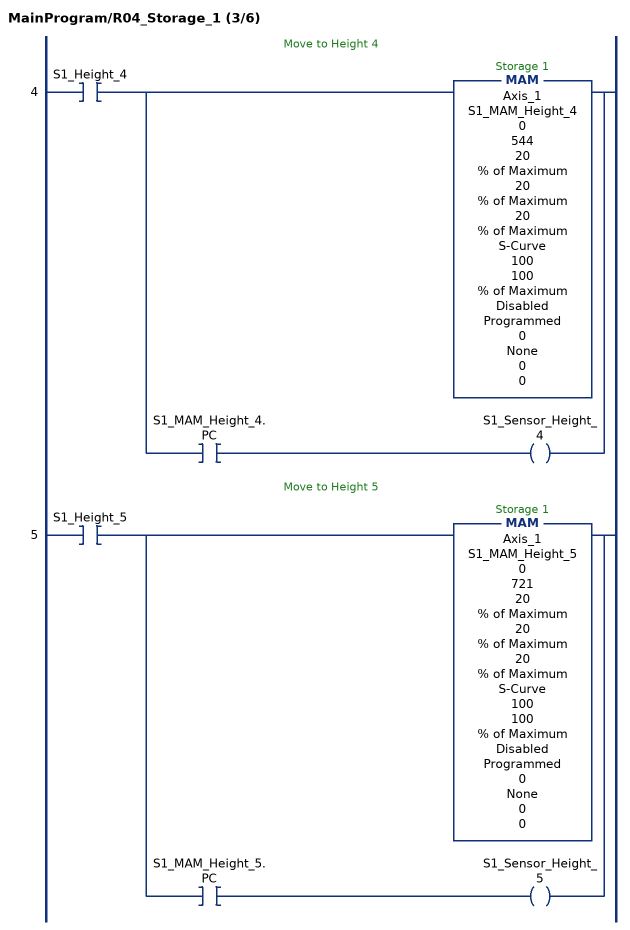
   // Move to Height 4
   4: XIC(S1_Height_4)[MAM(Axis_1,S1_MAM_Height_4,0,544,20,% of Maximum,20,% of Maximum,20,% of Maximum,S-Curve,100,100,% of Maximum,Disabled,Programmed,0,None,0,0) ,XIC(S1_MAM_Height_4.PC) OTE(S1_Sensor_Height_4) ];
   // Move to Height 5
   5: XIC(S1_Height_5)[MAM(Axis_1,S1_MAM_Height_5,0,721,20,% of Maximum,20,% of Maximum,20,% of Maximum,S-Curve,100,100,% of Maximum,Disabled,Programmed,0,None,0,0) ,XIC(S1_MAM_Height_5.PC) OTE(S1_Sensor_Height_5) ];
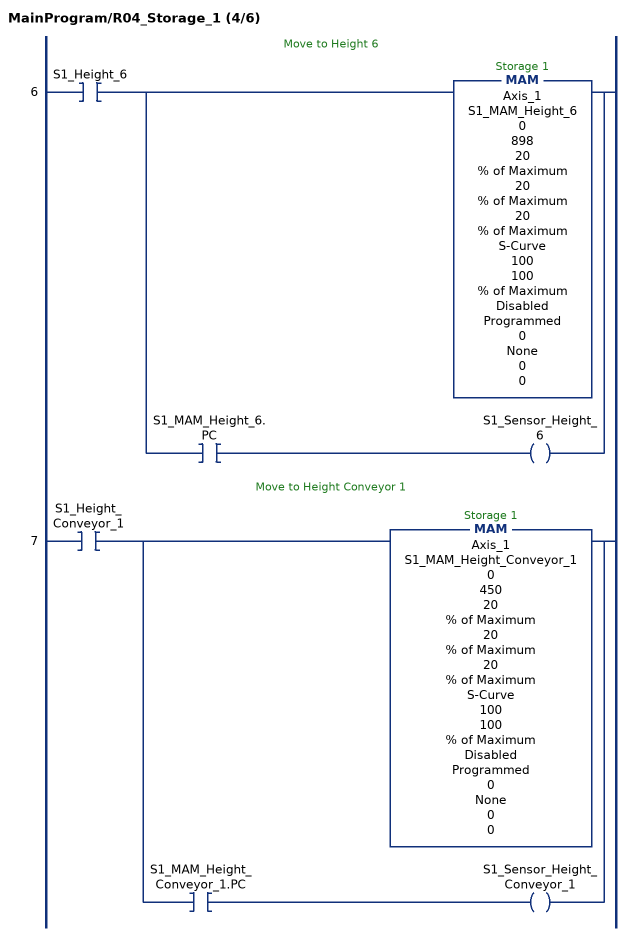
   // Move to Height 6
   6: XIC(S1_Height_6)[MAM(Axis_1,S1_MAM_Height_6,0,898,20,% of Maximum,20,% of Maximum,20,% of Maximum,S-Curve,100,100,% of Maximum,Disabled,Programmed,0,None,0,0) ,XIC(S1_MAM_Height_6.PC) OTE(S1_Sensor_Height_6) ];
   // Move to Height Conveyor 1
   7: XIC(S1_Height_Conveyor_1)[MAM(Axis_1,S1_MAM_Height_Conveyor_1,0,450,20,% of Maximum,20,% of Maximum,20,% of Maximum,S-Curve,100,100,% of Maximum,Disabled,Programmed,0,None,0,0) ,XIC(S1_MAM_Height_Conveyor_1.PC) OTE(S1_Sensor_Height_Conveyor_1) ];
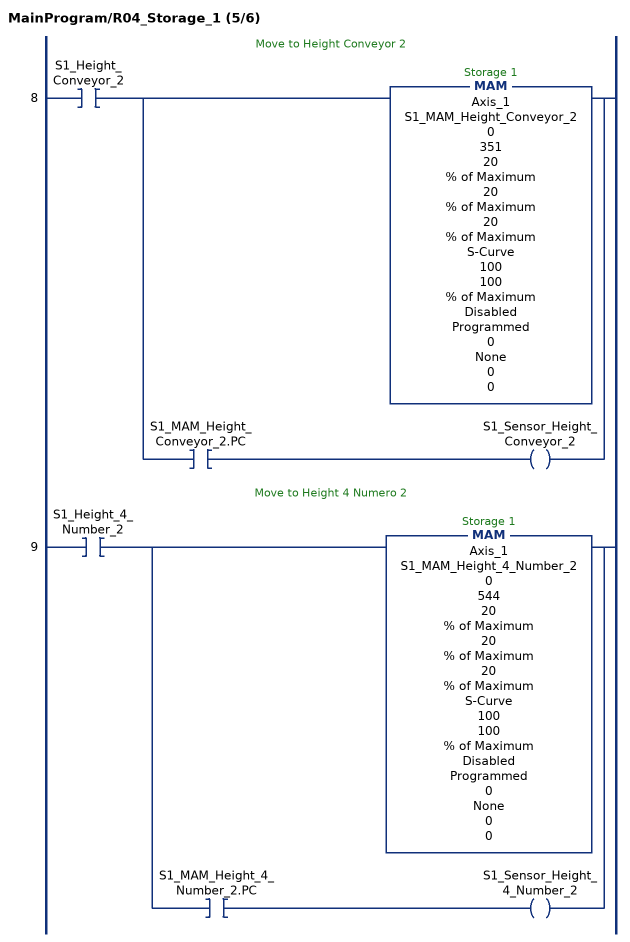
   // Move to Height Conveyor 2
   8: XIC(S1_Height_Conveyor_2)[MAM(Axis_1,S1_MAM_Height_Conveyor_2,0,351,20,% of Maximum,20,% of Maximum,20,% of Maximum,S-Curve,100,100,% of Maximum,Disabled,Programmed,0,None,0,0) ,XIC(S1_MAM_Height_Conveyor_2.PC) OTE(S1_Sensor_Height_Conveyor_2) ];
   // Move to Height 4 Numero 2
   9: XIC(S1_Height_4_Number_2)[MAM(Axis_1,S1_MAM_Height_4_Number_2,0,544,20,% of Maximum,20,% of Maximum,20,% of Maximum,S-Curve,100,100,% of Maximum,Disabled,Programmed,0,None,0,0) ,XIC(S1_MAM_Height_4_Number_2.PC) OTE(S1_Sensor_Height_4_Number_2) ];
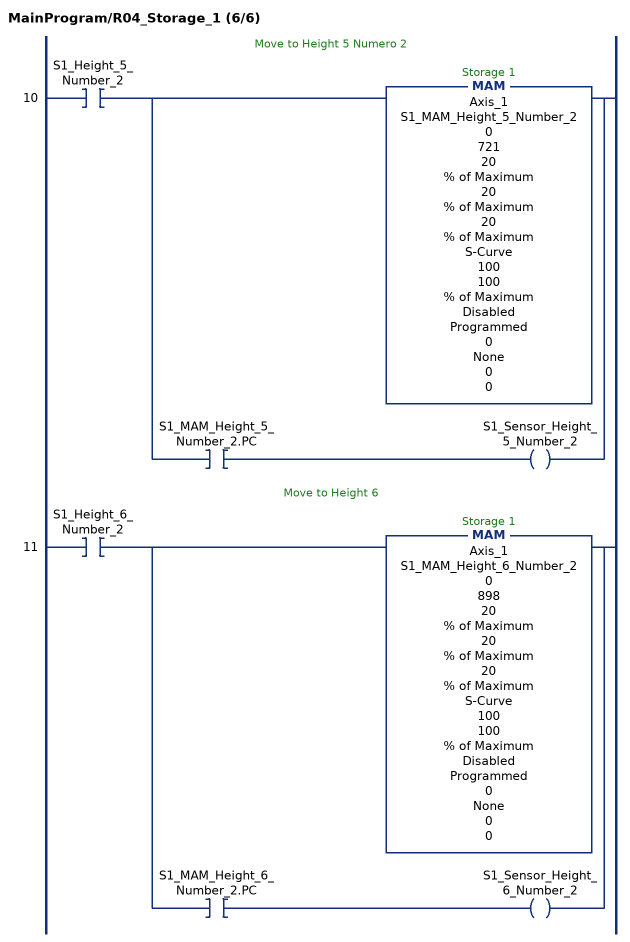
   // Move to Height 5 Numero 2
   10: XIC(S1_Height_5_Number_2)[MAM(Axis_1,S1_MAM_Height_5_Number_2,0,721,20,% of Maximum,20,% of Maximum,20,% of Maximum,S-Curve,100,100,% of Maximum,Disabled,Programmed,0,None,0,0) ,XIC(S1_MAM_Height_5_Number_2.PC) OTE(S1_Sensor_Height_5_Number_2) ];
   // Move to Height 6
   11: XIC(S1_Height_6_Number_2)[MAM(Axis_1,S1_MAM_Height_6_Number_2,0,898,20,% of Maximum,20,% of Maximum,20,% of Maximum,S-Curve,100,100,% of Maximum,Disabled,Programmed,0,None,0,0) ,XIC(S1_MAM_Height_6_Number_2.PC) OTE(S1_Sensor_Height_6_Number_2) ];
END_ROUTINE
